INTERFACE I_Disposable EXTENDS __SYSTEM.IQueryInterface

METHOD Dispose
END_METHOD

END_INTERFACE

(* stored: Version 1.1.0.1, ProductVersion 3.1.4024.9
   Itf I_Disposable: Id {ef8c751e-267f-45ec-babb-3d71f1bd95f8}
   Method Dispose: Id {1c7f6052-1eb0-490a-9cff-3be6b4764b89} *)
